PROGRAM Resetointivipu
VAR
	VALO1: BOOL;
	VALO2: BOOL;
	VALO3: BOOL;
END_VAR
VAR // added by the converter: edge detectors and wires of the graphical bodies
    _ft1, _ft2, _ft3 : F_TRIG;
END_VAR

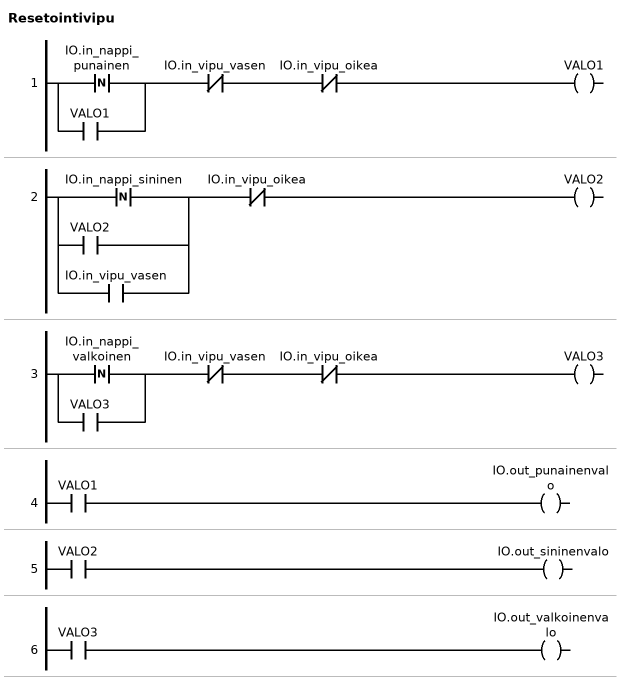
// NETWORK 1
_ft1(CLK := IO.in_nappi_punainen);
VALO1 := (_ft1.Q OR VALO1) AND NOT IO.in_vipu_vasen AND NOT IO.in_vipu_oikea;

// NETWORK 2
_ft2(CLK := IO.in_nappi_sininen);
VALO2 := (_ft2.Q OR VALO2 OR IO.in_vipu_vasen) AND NOT IO.in_vipu_oikea;

// NETWORK 3
_ft3(CLK := IO.in_nappi_valkoinen);
VALO3 := (_ft3.Q OR VALO3) AND NOT IO.in_vipu_vasen AND NOT IO.in_vipu_oikea;

// NETWORK 4
IO.out_punainenvalo := VALO1;

// NETWORK 5
IO.out_sininenvalo := VALO2;

// NETWORK 6
IO.out_valkoinenvalo := VALO3;

END_PROGRAM

(* stored: Version 1.1.0.1, ProductVersion 3.1.4024.10
   POU Resetointivipu: Id {89812091-e3ff-4526-93b0-418b13998916}, SpecialFunc None *)
